Omron CX-Programmer project NewProject (CX-Programmer 9.75)

# PLC NewPLC1: CP1L-E EM

## Global symbols (name address type ; comment)
C LedTimer
D StartProcess
DOL StartProcess

## Program NewProgram1 (cyclic task 0)
Local symbols
ANALOG_IN_1 A642 INT
ANALOG_READ D101 INT
ANLOG_0_10V D300 UINT_BCD
A_0 0.00 BOOL  ; reed
A_1 0.01 BOOL
A_CIL 100.00 BOOL
B_0 0.02 BOOL
B_1 0.03 BOOL
B_CIL_EN 200.09 BOOL
B_CIL_IN 100.02 BOOL
B_CIL_OUT 100.01 BOOL
C_0 0.04 BOOL
C_1 0.05 BOOL
C_CIL_EN 200.08 BOOL
C_CIL_IN 100.04 BOOL
C_CIL_OUT 100.03 BOOL
D_0 0.06 BOOL
D_1 0.07 BOOL
D_CIL 100.05 BOOL
EM_STOP 0.10 BOOL
FINISHED_TEACH_MODE 212.02 BOOL
GREEN_LED 100.07 BOOL
LED_BLINK_ENABLE 200.03 BOOL
PARAMETER_ADC D200 WORD
PROCESS 200.00 BOOL
RED_LED 101.00 BOOL
START_ENABLE 200.02 BOOL
START_PB 0.11 BOOL
STEP0 201.00 BOOL
STOP_PB 1.00 BOOL
TEACH_MODE 208.05 BOOL
TECH_FINISHED 209.14 BOOL
TECH_MODE 200.04 BOOL
TIMER 205.06 BOOL

### Section Program

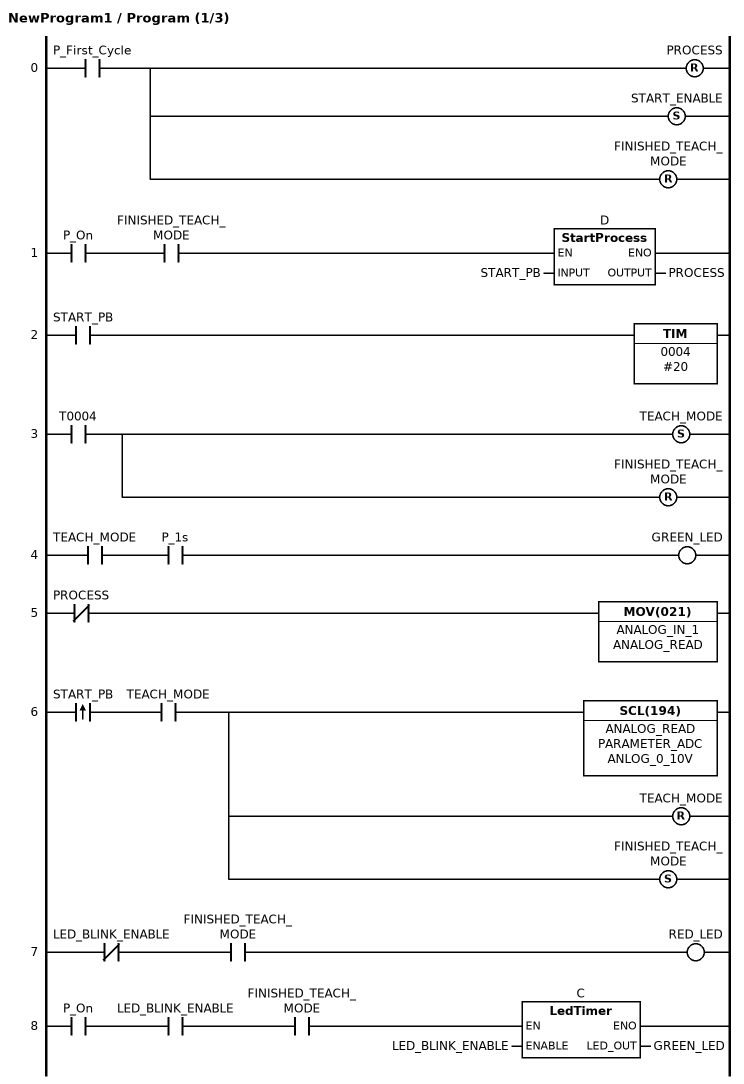
; rung 0
LD P_First_Cycle
RSET PROCESS
SET START_ENABLE
RSET FINISHED_TEACH_MODE
; rung 1
LD P_On
AND FINISHED_TEACH_MODE
CALL D : StartProcess (INPUT := START_PB, OUTPUT => PROCESS)
; rung 2
LD START_PB
TIM 0004 #20
; rung 3
LD T0004
SET TEACH_MODE
RSET FINISHED_TEACH_MODE
; rung 4
LD TEACH_MODE
AND P_1s
OUT GREEN_LED
; rung 5
LDNOT PROCESS
MOV(021) ANALOG_IN_1 ANALOG_READ
; rung 6
@LD START_PB
AND TEACH_MODE
SCL(194) ANALOG_READ PARAMETER_ADC ANLOG_0_10V
RSET TEACH_MODE
SET FINISHED_TEACH_MODE
; rung 7
LDNOT LED_BLINK_ENABLE
AND FINISHED_TEACH_MODE
OUT RED_LED
; rung 8
LD P_On
AND LED_BLINK_ENABLE
AND FINISHED_TEACH_MODE
CALL C : LedTimer (ENABLE := LED_BLINK_ENABLE, LED_OUT => GREEN_LED)

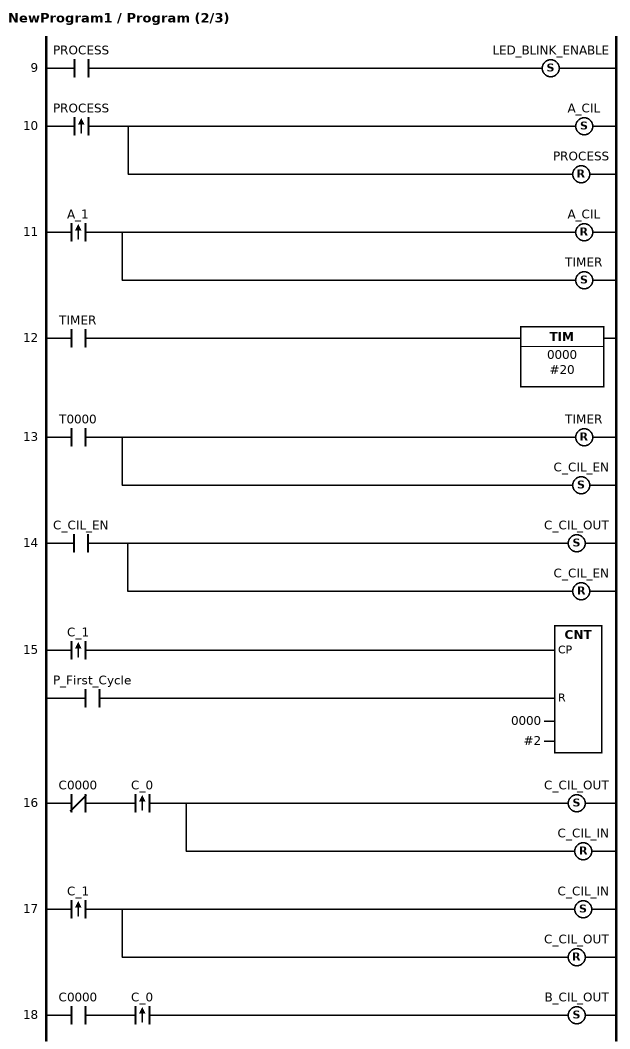
; rung 9
LD PROCESS
SET LED_BLINK_ENABLE
; rung 10
@LD PROCESS
SET A_CIL
RSET PROCESS
; rung 11
@LD A_1
RSET A_CIL
SET TIMER
; rung 12
LD TIMER
TIM 0000 #20
; rung 13
LD T0000
RSET TIMER
SET C_CIL_EN
; rung 14
LD C_CIL_EN
SET C_CIL_OUT
RSET C_CIL_EN
; rung 15
@LD C_1
LD P_First_Cycle
CNT 0000 #2
; rung 16
LDNOT C0000
@AND C_0
SET C_CIL_OUT
RSET C_CIL_IN
; rung 17
@LD C_1
SET C_CIL_IN
RSET C_CIL_OUT
; rung 18
LD C0000
@AND C_0
SET B_CIL_OUT

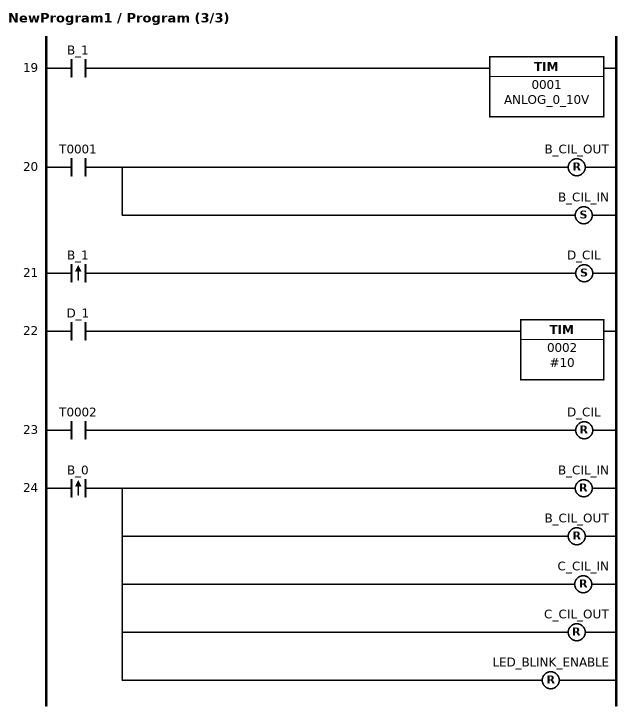
; rung 19
LD B_1
TIM 0001 ANLOG_0_10V
; rung 20
LD T0001
RSET B_CIL_OUT
SET B_CIL_IN
; rung 21
@LD B_1
SET D_CIL
; rung 22
LD D_1
TIM 0002 #10
; rung 23
LD T0002
RSET D_CIL
; rung 24
@LD B_0
RSET B_CIL_IN
RSET B_CIL_OUT
RSET C_CIL_IN
RSET C_CIL_OUT
RSET LED_BLINK_ENABLE

### Section END
; rung 0
END(001)

## Function block LedTimer
VAR_INPUT
  ENABLE : BOOL;
END_VAR
VAR_OUTPUT
  LED_OUT : BOOL;
END_VAR
VAR
  LED_BLINK_STATE : BOOL;
  ON_TIMER : TIMER;
  OFF_TIMER : TIMER;
END_VAR

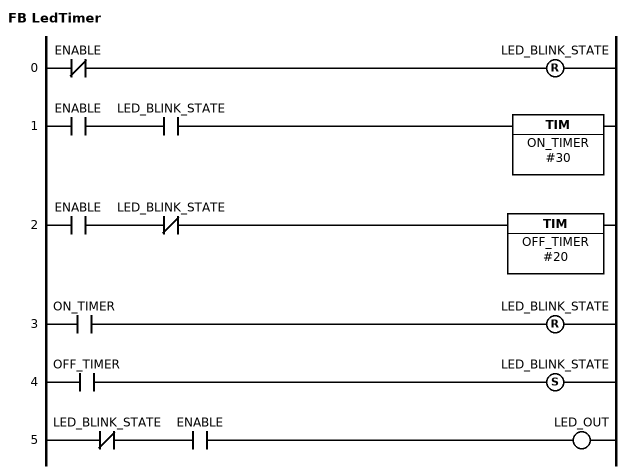
; rung 0
LDNOT ENABLE
RSET LED_BLINK_STATE
; rung 1
LD ENABLE
AND LED_BLINK_STATE
TIM ON_TIMER #30
; rung 2
LD ENABLE
ANDNOT LED_BLINK_STATE
TIM OFF_TIMER #20
; rung 3
LD ON_TIMER
RSET LED_BLINK_STATE
; rung 4
LD OFF_TIMER
SET LED_BLINK_STATE
; rung 5
LDNOT LED_BLINK_STATE
AND ENABLE
OUT LED_OUT

## Function block StartProcess
VAR_INPUT
  INPUT : BOOL;
END_VAR
VAR_OUTPUT
  OUTPUT : BOOL;
END_VAR
VAR
  TIMER0 : TIMER;
  COUNTER0 : COUNTER;
  PRESS_ONCE : BOOL;
END_VAR

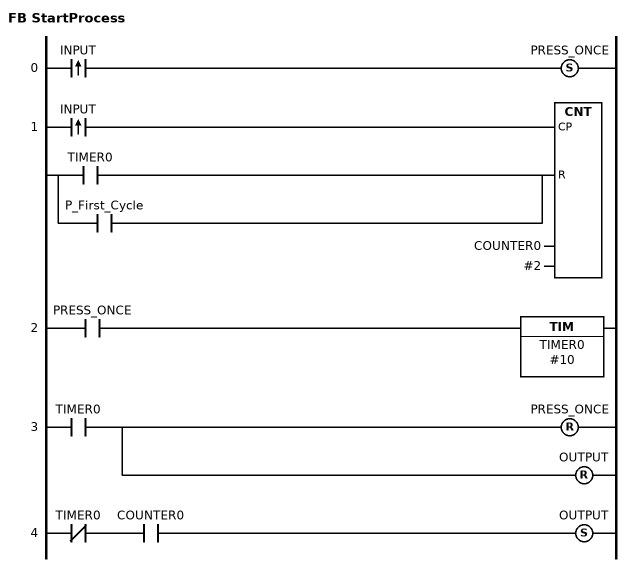
; rung 0
@LD INPUT
SET PRESS_ONCE
; rung 1
@LD INPUT
LD TIMER0
OR P_First_Cycle
CNT COUNTER0 #2
; rung 2
LD PRESS_ONCE
TIM TIMER0 #10
; rung 3
LD TIMER0
RSET PRESS_ONCE
RSET OUTPUT
; rung 4
LDNOT TIMER0
AND COUNTER0
SET OUTPUT